(* PLC project Unnamed, Unknown Unnamed 1 *)
(* stored: creationDateTime 2025-11-04T13:47:54, modificationDateTime 2025-11-04T13:57:15 *)

PROGRAM TONExample
  VAR
    Q_LED : BOOL := False;
    T_1 : TON;
    T_2 : TON;
    Flash_Period : TIME := T#1s;
  END_VAR

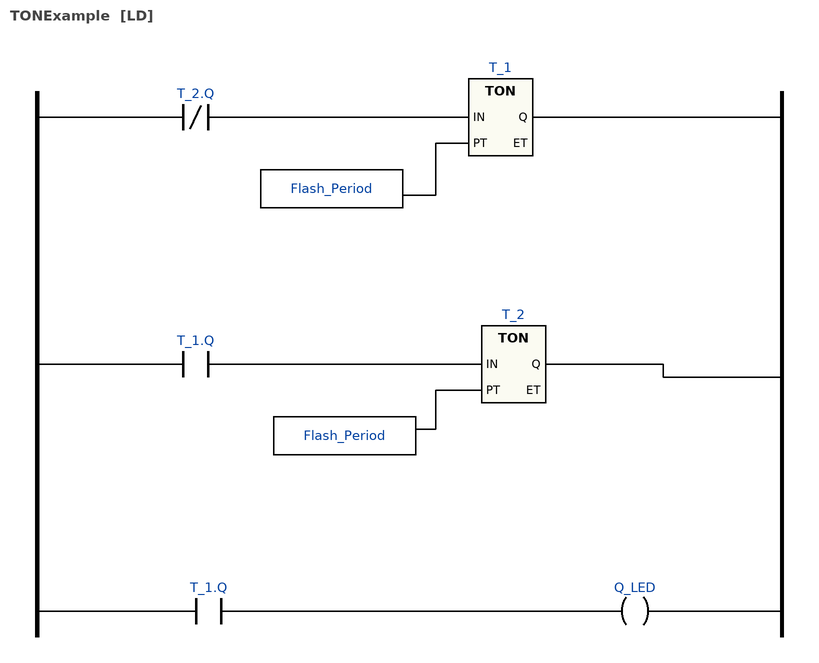
(* LD diagram, written out as Structured Text *)
Q_LED := T_1.Q;
T_1(IN := NOT T_2.Q, PT := Flash_Period);
T_2(IN := T_1.Q, PT := Flash_Period);
END_PROGRAM

PROGRAM TONTOFExample
  VAR
    Q_LED : BOOL := False;
    F_LEDON : BOOL := False;
    TON0 : TON;
    TOF0 : TOF;
    FlashTime : TIME := T#1s;
  END_VAR

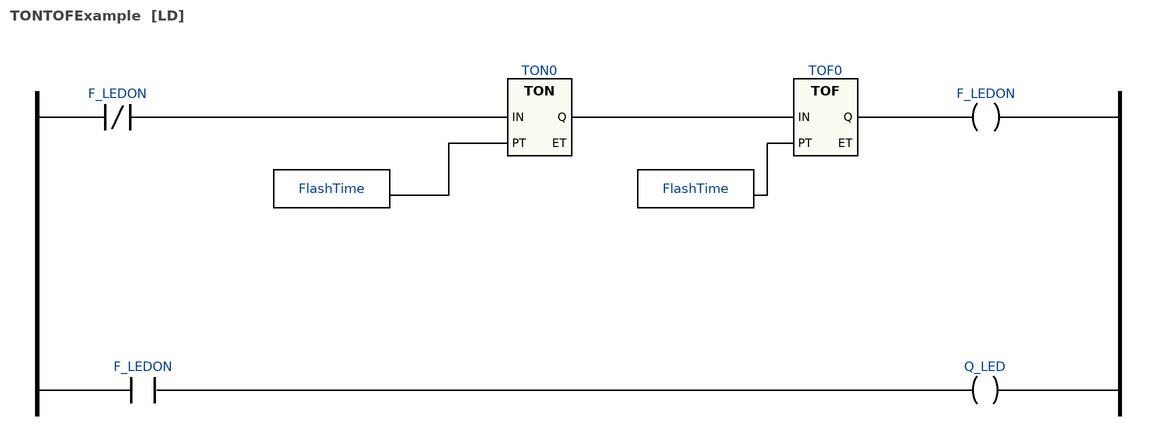
(* LD diagram, written out as Structured Text *)
TON0(IN := NOT F_LEDON, PT := FlashTime);
TOF0(IN := TON0.Q, PT := FlashTime);
F_LEDON := TOF0.Q;
Q_LED := F_LEDON;
END_PROGRAM

CONFIGURATION Config0
  RESOURCE Res0 ON PLC
    TASK task0(INTERVAL := T#20ms, PRIORITY := 0);
    PROGRAM instance0 WITH task0 : TONExample;
    PROGRAM instance1 WITH task0 : TONTOFExample;
  END_RESOURCE
END_CONFIGURATION
